ABB RobotStudio station: loading_area_main.rsstn

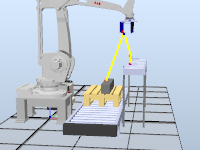
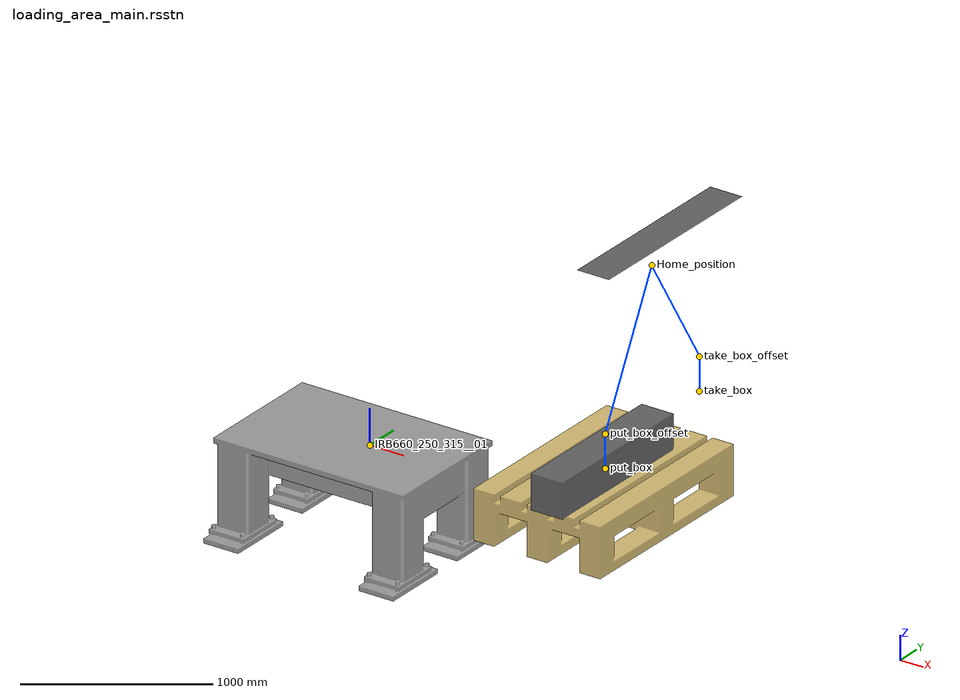
[picture v1: parts stored in the station drawn from their meshes, with robot base, taught points and paths (robot models come from the ABB library and are not in the file)]
Station Solution4 (saved by RobotStudio 21.2.9526.0)
Controller IRB660_250_315
  mechanical unit ROB_1: IRB660_250_315__01, 6 joints, base frame (0, 0, 570) mm
Layout (positions relative to the parent item):
  - IRB660_250_315__01 [mechanism, from Robots\IRB660_250_315__01.rslib] at (0, 0, 570) mm; joint values [0, 0, 0, 0] (rad or m)
  - conv_box_top [part, from библиотеки\conv_box_top.rslib] at (1800, -500, 1316.27) mm
  - conv_pallets_top [part, from библиотеки\conv_pallets_top.rslib] at (800, 2460, 435) mm
  - IRC5_Control-Module [part, from Equipment\IRC5_Control-Module.rslib] at (105.41, 1247.41, 100) mm, rotated rx 90 ry 0 rz 90 deg
  - Стол_2 [part] at (445, -335, 540) mm, rotated rx 90 ry 0 rz 90 deg, size 980 x 570 x 1200 mm
  - Box_200 [part] at (1299.16, -404, 933) mm, rotated rx 0 ry 90 rz 0 deg, size 210 x 1000 x 200 mm
  - pallet [part] at (1700, -350, 415) mm, rotated rx 0 ry -90 rz 0 deg, size 298 x 1200 x 800 mm
  - My_Gripper [mechanism] at (1910, 0, 2403) mm, rotated rx 180 ry 0 rz 180 deg; joint values [-0.0498] (rad or m)
      TCP My_Gripper_1 at (178, -180, 244) mm
      links: L1, L2
  - Attacher [part] at (1734, -605, 2307) mm, rotated rx 0 ry 90 rz 0 deg, size 0 x 1200 x 200 mm
Attachment: My_Gripper is attached to IRB660_250_315__01 / Link6
Attachment: Attacher is attached to IRB660_250_315__01 / Link6
EventTableEntry 1190: Group=, Trigger=doOpenGripper 1191, Actions=[EventTableActionMechanicalPose 1192], Comment=, ActivationMode=2, Cyclic=false
EventTableTriggerIO 1191: IOValue=[1], IRC5Controller=? -1, Operator=0, SignalSource=IRB660_250_315 515
EventTableActionMechanicalPose 1192: VirtualSignal=, Mechanism=My_Gripper 1033, ToPoseName=HomePosition, VirtualSignalValue=[1]
EventTableEntry 1193: Group=, Trigger=doCloseGripper 1194, Actions=[EventTableActionMechanicalPose 1195], Comment=, ActivationMode=2, Cyclic=false
EventTableTriggerIO 1194: IOValue=[1], IRC5Controller=? -1, Operator=0, SignalSource=IRB660_250_315 515
EventTableActionMechanicalPose 1195: VirtualSignal=, Mechanism=My_Gripper 1033, ToPoseName=Pose Closed, VirtualSignalValue=[1]
EventTableEntry 1199: Group=, Trigger=Attach 1200, Actions=[EventTableActionAttach 1201], Comment=, ActivationMode=2, Cyclic=false
EventTableTriggerIO 1200: IOValue=[1], IRC5Controller=? -1, Operator=0, SignalSource=IRB660_250_315 515
EventTableActionAttach 1201: AttachmentParent=Attacher 1197, AttachmentChild=Box_200 1016, MountObject=true, Offset=[X=1, Y=0, Z=0, W=0, X=0, Y=1, Z=0, W=0, X=0, Y=0, Z=1, W=0, X=0, Y=0, Z=0, W=1], FlangeIndext=0, FindNearest=false
EventTableEntry 1202: Group=, Trigger=Detach 1203, Actions=[EventTableActionDetach 1204], Comment=, ActivationMode=2, Cyclic=false
EventTableTriggerIO 1203: IOValue=[1], IRC5Controller=? -1, Operator=0, SignalSource=IRB660_250_315 515
EventTableActionDetach 1204: AttachmentParent=Attacher 1197, AttachmentChild=Box_200 1016
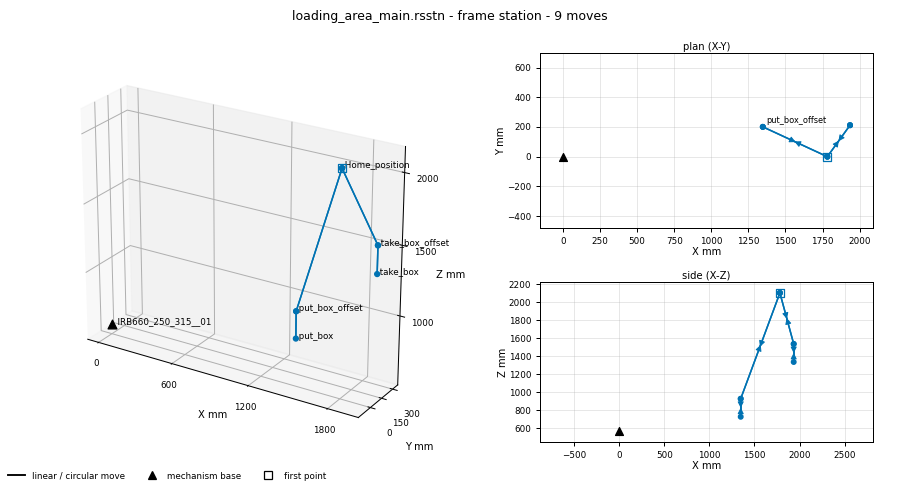
[picture p0: tool path of loading_area_main.rsstn in frame station, 9 of 9 moves have a stored position in this frame; points joined in program order, loops and branches not executed]
Targets, tools, work objects and paths stored in the station, written as RAPID:
! task T_ROB1
MODULE CalibData
  PERS tooldata My_Gripper_1:=[TRUE,[[128.15625,0,299],[1,0,0,0]],[2.5,[0,0,100],[1,0,0,0],0,0,0]];
  TASK PERS wobjdata Wobj_box:=[FALSE,TRUE,"",[[0,0,0],[1,0,0,0]],[[0,0,0],[1,0,0,0]]];
  TASK PERS wobjdata Wobj_pallet:=[FALSE,TRUE,"",[[0,0,0],[1,0,0,0]],[[0,0,0],[1,0,0,0]]];
ENDMODULE

! task T_ROB1
MODULE Module1
  CONST robtarget take_box:=[[1935,212,1338],[0,0,1,0],[0,0,0,0],[9E+09,9E+09,9E+09,9E+09,9E+09,9E+09]];
  CONST robtarget put_box:=[[1347,201,730],[0,0,1,0],[0,0,0,0],[9E+09,9E+09,9E+09,9E+09,9E+09,9E+09]];
  CONST robtarget take_box_offset:=[[1935,212,1538],[0,0,1,0],[0,0,0,0],[9E+09,9E+09,9E+09,9E+09,9E+09,9E+09]];
  CONST robtarget put_box_offset:=[[1347,201,930],[0,0,1,0],[0,0,0,0],[9E+09,9E+09,9E+09,9E+09,9E+09,9E+09]];
  CONST robtarget Home_position:=[[1781.84375,0,2104],[0,0,1,0],[0,0,0,0],[9E+09,9E+09,9E+09,9E+09,9E+09,9E+09]];
  PROC Path_10()
    MoveL Home_position,v1000,z100,My_Gripper_1\WObj:=wobj0;
    MoveL take_box_offset,v1000,z100,My_Gripper_1\WObj:=Wobj_box;
    MoveL take_box,v1000,z100,My_Gripper_1\WObj:=Wobj_box;
    MoveL take_box_offset,v1000,z100,My_Gripper_1\WObj:=Wobj_box;
    MoveL Home_position,v1000,z100,My_Gripper_1\WObj:=wobj0;
    MoveL put_box_offset,v1000,z100,My_Gripper_1\WObj:=Wobj_pallet;
    MoveL put_box,v1000,z100,My_Gripper_1\WObj:=Wobj_pallet;
    MoveL put_box_offset,v1000,z100,My_Gripper_1\WObj:=Wobj_pallet;
    MoveL Home_position,v1000,z100,My_Gripper_1\WObj:=wobj0;
  ENDPROC
ENDMODULE

